{attribute 'linkalways'} 
{attribute 'no_explicit_call' := 'This FB is a CLASS and must be accessed using methods or properties'}
{attribute 'enable_dynamic_creation'}
FUNCTION_BLOCK Node_F_VN_GetAt_TcVnVector2_REAL EXTENDS VisionNode
VAR
    ipContainer : _ITcVnContainer;
    aElement : _TcVnVector2_REAL;
    nIndex : _ULINT(0);
    hrPrev : _HRESULT(S_OK);
    hresult : _HRESULT(S_OK);
END_VAR

METHOD PUBLIC  Clone : I_Node
VAR
	pNode : POINTER TO Node_F_VN_GetAt_TcVnVector2_REAL;
END_VAR
pNode := __NEW(Node_F_VN_GetAt_TcVnVector2_REAL);
Clone := pNode^;
END_METHOD

METHOD FB_init : BOOL
VAR_INPUT
	bInitRetains : BOOL; // if TRUE, the retain variables are initialized (warm start / cold start)
	bInCopyCode : BOOL;  // if TRUE, the instance afterwards gets moved into the copy code (online change)
END_VAR
AddInput('ipContainer', ipContainer);
AddParameter('nIndex', nIndex);
AddInput('hrPrev', hrPrev);
AddOutput('aElement', aElement);
AddOutput('hresult',hresult);
END_METHOD

METHOD PROTECTED OnExecute
hresult.Value := F_VN_GetAt_TcVnVector2_REAL(
    ipContainer := ipContainer.Value,
    aElement := aElement.Value,
    nIndex := nIndex.Value,
    hrPrev:= hrPrev.Value);
END_METHOD

METHOD PUBLIC PreExecutionCheck
VAR_INPUT
	Check : I_PreExecutionChecks;
END_VAR
Check.IsTrue(ipContainer.IsValid, 'ipContainer must be a valid container');
Check.IsTrue(ipContainer.IsType(TC_GLOBAL_CONST_LIST.ContainerType_Vector_TcVnVector2_REAL), 'ipContainer contains incorrect type');
END_METHOD

END_FUNCTION_BLOCK

(* stored: Version 1.1.0.1, ProductVersion 3.1.4026.13
   POU Node_F_VN_GetAt_TcVnVector2_REAL: Id {afa8333e-acb7-494d-a969-1ef6d2f8bf0a}, SpecialFunc None
   Folder Constructor: Id {8862b3d0-660e-4c6d-9aaa-64674bdcdb4a}
   Method Clone: Id {8a687c59-fef8-4da3-9afa-006f31253975}
   Method FB_init: Id {86246899-b03c-4897-ab9b-229a5d56bb8f}
   Method OnExecute: Id {091b4f77-2400-4442-a31d-0db19c091042}
   Method PreExecutionCheck: Id {78cdf421-6419-4f55-8d7c-28b35e8adc6f} *)
